(* PLC project Unnamed, Unknown Unnamed 1 *)
(* stored: creationDateTime 2023-12-24T17:42:03, modificationDateTime 2023-12-26T23:56:32 *)

PROGRAM FrequencyCounter
  VAR
    Frequency_In AT %IX0.0 : BOOL;  (* Process Variable input in frequency. *)
    Frequency_Value AT %QW0 : UINT;
  END_VAR
  VAR
    Clock : BOOL;  (* Clock generator for the frequency counter. *)
    TON0 : TON;
    CTU0 : CTU;
    F_Aux_00 : INT;
    F_Aux_01 : INT;
    F_Aux_02 : INT;
    F_Aux_03 : INT;
    F_SUM : INT;
    F_AVERAGE : REAL;
    F_TRIG0 : F_TRIG;
    R_TRIG0 : R_TRIG;
    CTU1 : CTU;
    F_TRIG1 : F_TRIG;
    R_TRIG1 : R_TRIG;
  END_VAR
  VAR  (* added by the conversion: wires and edge detectors of the diagram *)
    R_TRIG1_2 : R_TRIG;
    R_TRIG2 : R_TRIG;
  END_VAR

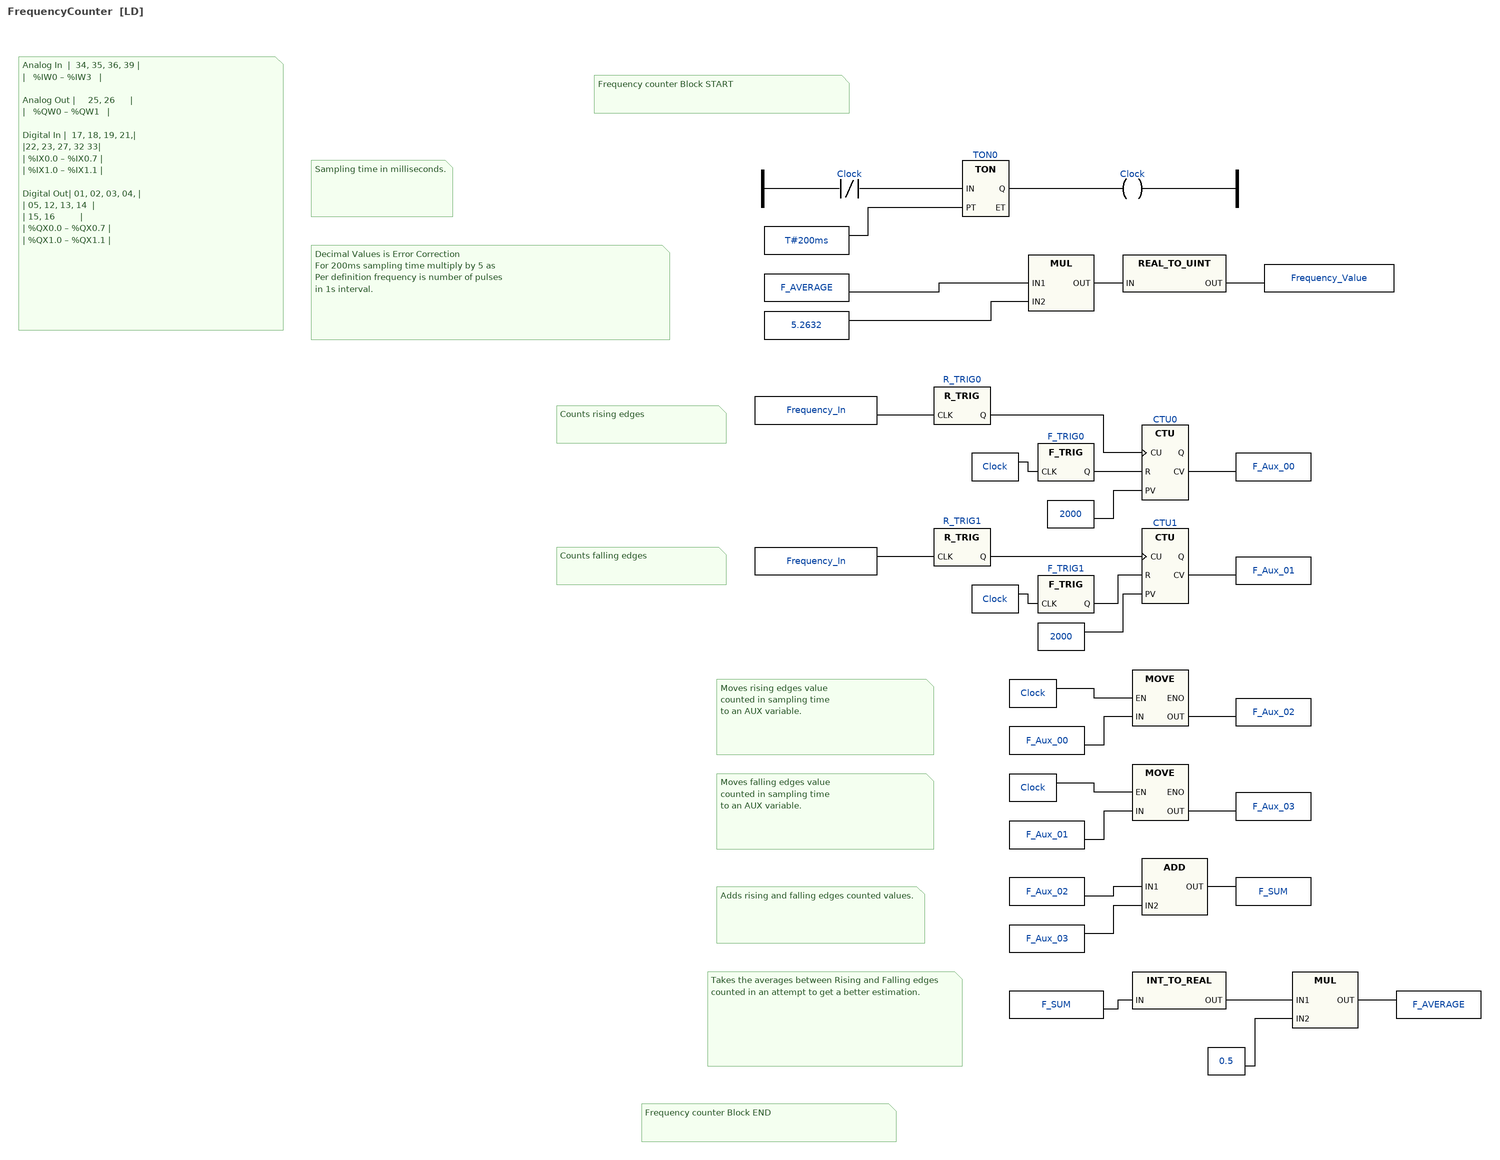
(* LD diagram, written out as Structured Text *)
(* Analog In  |  34, 35, 36, 39 |
           |   %IW0 – %IW3   |

Analog Out |     25, 26      |
           |   %QW0 – %QW1   |

Digital In |  17, 18, 19, 21,|
           |22, 23, 27, 32 33|
           | %IX0.0 – %IX0.7 |
           | %IX1.0 – %IX1.1 |

Digital Out| 01, 02, 03, 04, |
           | 05, 12, 13, 14  |
           | 15, 16          |
           | %QX0.0 – %QX0.7 |
           | %QX1.0 – %QX1.1 | *)
(* Frequency counter Block START *)
(* Sampling time in milliseconds. *)
TON0(IN := NOT Clock, PT := T#200ms);
Clock := TON0.Q;
(* Decimal Values is Error Correction
For 200ms sampling time multiply by 5 as
Per definition frequency is number of pulses
in 1s interval. *)
Frequency_Value := REAL_TO_UINT(F_AVERAGE * 5.2632);
(* Counts rising edges *)
R_TRIG0(CLK := Frequency_In);
R_TRIG1_2(CLK := R_TRIG0.Q);
F_TRIG0(CLK := Clock);
CTU0(CU := R_TRIG1_2.Q, R := F_TRIG0.Q, PV := 2000);
F_Aux_00 := CTU0.CV;
(* Counts falling edges *)
R_TRIG1(CLK := Frequency_In);
R_TRIG2(CLK := R_TRIG1.Q);
F_TRIG1(CLK := Clock);
CTU1(CU := R_TRIG2.Q, R := F_TRIG1.Q, PV := 2000);
F_Aux_01 := CTU1.CV;
(* Moves rising edges value
counted in sampling time
to an AUX variable. *)
IF Clock THEN F_Aux_02 := F_Aux_00; END_IF;
(* Moves falling edges value
counted in sampling time
to an AUX variable. *)
IF Clock THEN F_Aux_03 := F_Aux_01; END_IF;
F_SUM := F_Aux_02 + F_Aux_03;
(* Adds rising and falling edges counted values. *)
(* Takes the averages between Rising and Falling edges counted in an attempt to get a better estimation. *)
F_AVERAGE := INT_TO_REAL(F_SUM) * 0.5;
(* Frequency counter Block END *)
END_PROGRAM

CONFIGURATION Config0
  RESOURCE Res0 ON PLC
    TASK task0(INTERVAL := T#0.5ms, PRIORITY := 0);
    PROGRAM instance0 WITH task0 : FrequencyCounter;
  END_RESOURCE
END_CONFIGURATION
